Staubli VAL3: cycle_isPause.pgx

program cycle_isPause(bool& x_bPause[] (dimensions=1))
begin
  //
  // ask for pause status
  //
  x_bPause=cycleStatus:bPause
end
